% RSLogix 500 project Counters.RSS, saved by version 8.30.00.16 %
PROJECT "LEC24"    % processor: Bul.1763 MicroLogix 1100 Series B %

PROGRAM FILES
  LAD 2   7 rungs

DATA FILES
  O0 OUTPUT  4 elements
  I1 INPUT  6 elements
  S2 STATUS  66 elements
  B3 BINARY  1 elements
  T4 TIMER  1 elements
  C5 COUNTER  2 elements
  R6 CONTROL  1 elements
  N7 INTEGER  1 elements
  F8 FLOAT  1 elements

LADDER 2
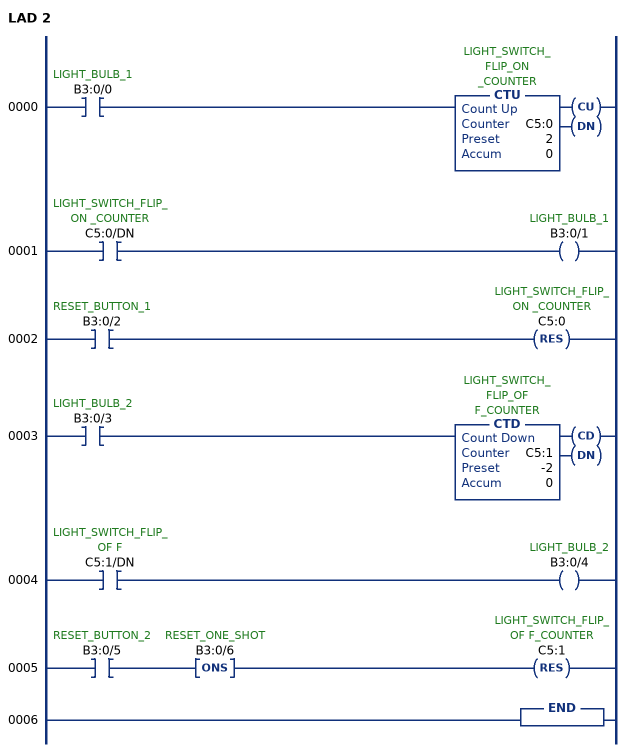
% Rung: 0 %
SOR XIC B3:0/0 CTU C5:0 2 0 EOR
%   B3:0/0  "LIGHT_BULB_1" %
%   C5:0  "LIGHT_SWITCH_FLIP_ON _COUNTER" %
% Rung: 1 %
SOR XIC C5:0/DN OTE B3:0/1 EOR
%   C5:0/DN  "LIGHT_SWITCH_FLIP_ON _COUNTER" %
%   B3:0/1  "LIGHT_BULB_1" %
% Rung: 2 %
SOR XIC B3:0/2 RES C5:0 EOR
%   B3:0/2  "RESET_BUTTON_1" %
%   C5:0  "LIGHT_SWITCH_FLIP_ON _COUNTER" %
% Rung: 3 %
SOR XIC B3:0/3 CTD C5:1 -2 0 EOR
%   B3:0/3  "LIGHT_BULB_2" %
%   C5:1  "LIGHT_SWITCH_FLIP_OF F_COUNTER" %
% Rung: 4 %
SOR XIC C5:1/DN OTE B3:0/4 EOR
%   C5:1/DN  "LIGHT_SWITCH_FLIP_OF F" %
%   B3:0/4  "LIGHT_BULB_2" %
% Rung: 5 %
SOR XIC B3:0/5 ONS B3:0/6 RES C5:1 EOR
%   B3:0/5  "RESET_BUTTON_2" %
%   B3:0/6  "RESET_ONE_SHOT" %
%   C5:1  "LIGHT_SWITCH_FLIP_OF F_COUNTER" %
% Rung: 6 %
SOR END EOR

DATA TABLE (non-zero values as saved)
DATA C5
% .PRE .ACC %
% C5:0 % 2 0
% C5:1 % -2 0
